PROGRAM MAIN
VAR
    Initialize	:	BOOL := TRUE;

    fbLogHandler : FB_LogHandler;
    fbEcatDiag : FB_EcatDiagWrapper;

    {attribute 'pytmc' := '
    pv: @(PREFIX)BeamParamCntl
    '}
    fbBPControl : FB_BPControlDevice(nID:=10);
	
	PERanges : PE_Ranges;
	{attribute 'TcLinkTo' := 'TIIB[PMPS_Premp]^Channel 8^Output;'}
	bM1K1_OUT_Override AT %Q* : BOOL; // Using this book to completely overrule the last bit of the BC interface.
	
	//System Time
	 {attribute 'pytmc' := '
        pv: @(PREFIX)SystemDT
        io: i
     '}
	SystemTime:DINT;
	fbTime : FB_LocalSystemTime := ( bEnable := TRUE, dwCycle := 1 ); //Get current system time, used for override
	fbTime_to_UTC: FB_TzSpecificLocalTimeToSystemTime;
	fbGetTimeZone: FB_GetTimeZoneInformation;
END_VAR

//Arbiter PLC

IF Initialize THEN
    Initialize := FALSE;
END_IF

// Ethercat Diagnostics
fbEcatDiag();

// PMPS Functionality
CurrentBPUpdate();

///////////////////////////////////////////////////
// This code should be disabled or removed in deployment
// Might have a switch to change to simulation mode
MachineSimulation();
//Testing();
///////////////////////////////////////////////////

// Dummy device for controling pmps beam parameters
fbBPControl(Arbiter:=g_fbArbiter1);



PMPS_Arbiter();

P_AT1K0_SL1K0();

bM1K1_OUT_Override := PMPS_GVL.stCurrentBeamParameters.aVetoDevices[PMPS.K_Stopper.MR1K1_OUT];

fbLogHandler();
A_SystemTime();
Fast_Faults_Evaluate();

ACTION A_SystemTime:
//Get local System Time
fbTime(sNetID:='');
//Get Time Zone
fbGetTimeZone(sNetID:='',bExecute:=TRUE,tTimeout:=T#10S);
//change local time to UTC to be compatible with unix time epoch widget
fbTime_to_UTC(in:= fbTime.systemTime , tzInfo:=fbGetTimeZone.tzInfo);

SystemTime:= TO_DINT(TO_DT(SystemTime_TO_DT(fbTime_to_UTC.out)));
END_ACTION

ACTION Initialize:

END_ACTION

END_PROGRAM

(* stored: Version 1.1.0.1, ProductVersion 3.1.4022.18
   POU MAIN: Id {8a7bcfd2-1a2b-4363-aa47-c19391bf1f9c}, SpecialFunc None
   Action A_SystemTime: Id {932b887a-aeb4-43ef-9b71-03a84b8275c9}
   Action Initialize: Id {b0ee480a-3d4b-001d-04c4-43cdc47895c8} *)
